Staubli VAL3: onF3Event.pgx

program onF3Event()
  local string l_sMessage
  local string l_sItem
begin

     // load the page AXIS8


end
